{attribute 'qualified_only'}
{attribute 'strict'}
{attribute 'to_string'}
TYPE eBetriebszustand :
(
	Off        := 0,   // nicht betriebsbereit
	Error      := 1,   // Fehlerbehafteter Stop
	Setup      := 2,   // Wartung
	Warning    := 3,   // nicht fehlerbehafteter, nicht geplanter Stop
	Init       := 4,   // Herstellung Betriebsbereitschaft
	Ready      := 5,   // betriebsbereit
	Production := 6,   // Betrieb
	Done       := 7,   // Betrieb abgeschlossen
	Stop       := 8
);
END_TYPE

(* stored: Version 1.1.0.1, ProductVersion 3.1.4026.18
   DUT eBetriebszustand: Id {63ba0446-c3a7-491d-b3d6-801e92b1dc47} *)
